Universal Robots PolyScope program: IAC002 PathMove.urp

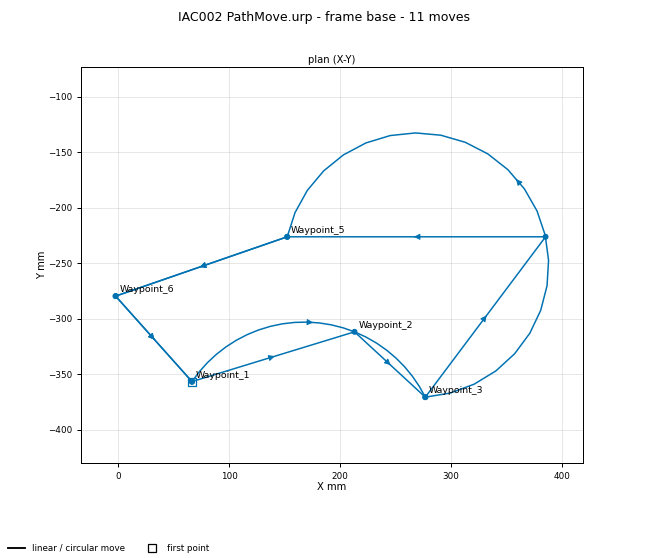
[picture p0: tool path of IAC002 PathMove.urp in frame base, 11 of 13 moves have a stored position in this frame; points joined in program order, loops and branches not executed]
Program IAC002 PathMove (installation=default directory=/programs createdIn=5.9.1.1031110 lastSavedIn=5.9.1.1031110 robotSerialNumber=20195501059)
Calibrated DH parameters: a=[0.000146, -0.418764, -0.053981, 0.000058, -0.000023, 0]; d=[0.162545, 37.319448, -206.067439, 168.881546, 0.09955, 0.099464]; alpha=[1.57004, -0.001979, 0.002304, 1.570607, -1.57066, 0]; deltaTheta=[0, -0.174616, -1.258233, 1.432844, -0.000001, 0]
Robot Program (runOnlyOnce=false)
  MoveP speed 100 mm/s, acceleration 1200 mm/s^2 (blendRadius=0.025 useActiveTCP=true) feature=Base
    Waypoint Waypoint_1: TCP in base x=66.517 y=-356.748 z=9.401 mm, rx=0.8699 ry=3.0055 rz=-0.0545 rad; joints [78.529, -92.143, 143.844, -143.739, 270.633, 20.88] deg; TCP offset x=0 y=0 z=174 mm, rx=0 ry=0 rz=0 rad
    Waypoint Waypoint_2: TCP in base x=212.953 y=-311.931 z=9.413 mm, rx=0.8699 ry=3.0054 rz=-0.0546 rad; joints [103.909, -89.736, 141.52, -143.858, 269.699, 46.246] deg
    Waypoint Waypoint_3: TCP in base x=276.697 y=-370.783 z=9.413 mm, rx=0.8699 ry=3.0055 rz=-0.0545 rad; joints [110.314, -78.862, 128.784, -141.938, 269.445, 52.645] deg
    Waypoint Waypoint_4: TCP in base x=385.033 y=-226.321 z=9.405 mm, rx=0.8698 ry=3.0055 rz=-0.0546 rad; joints [133, -80.507, 130.77, -141.882, 268.715, 75.321] deg
    Waypoint Waypoint_5: TCP in base x=152.305 y=-226.334 z=9.423 mm, rx=0.8699 ry=3.0055 rz=-0.0546 rad; joints [94.734, -109.57, 155.879, -138.422, 270.064, 37.053] deg
    Waypoint Waypoint_6: TCP in base x=-2.245 y=-279.765 z=9.416 mm, rx=0.8699 ry=3.0055 rz=-0.0546 rad; joints [59.76, -108.29, 155.126, -138.596, 271.286, 2.1] deg
    Waypoint Waypoint_1: TCP in base x=66.517 y=-356.748 z=9.401 mm, rx=0.8699 ry=3.0055 rz=-0.0545 rad; joints [78.529, -92.143, 143.844, -143.739, 270.633, 20.88] deg
  MoveP speed 150 mm/s, acceleration 1200 mm/s^2 (blendRadius=0.025 useActiveTCP=true) feature=Base
    CircleMove (OrientationMode=FIXED)
      Waypoint Waypoint_2: TCP in base x=212.953 y=-311.931 z=9.413 mm, rx=0.8699 ry=3.0054 rz=-0.0546 rad; joints [103.909, -89.736, 141.52, -143.858, 269.699, 46.246] deg
      Waypoint Waypoint_3: TCP in base x=276.697 y=-370.783 z=9.413 mm, rx=0.8699 ry=3.0055 rz=-0.0545 rad; joints [110.314, -78.862, 128.784, -141.938, 269.445, 52.645] deg
    CircleMove (OrientationMode=UNCONSTRAINED)
      Waypoint Waypoint_4: TCP in base x=385.033 y=-226.321 z=9.405 mm, rx=0.8698 ry=3.0055 rz=-0.0546 rad; joints [133, -80.507, 130.77, -141.882, 268.715, 75.321] deg
      Waypoint Waypoint_5: TCP in base x=152.305 y=-226.334 z=9.423 mm, rx=0.8699 ry=3.0055 rz=-0.0546 rad; joints [94.734, -109.57, 155.879, -138.422, 270.064, 37.053] deg
    Waypoint Waypoint_6: TCP in base x=-2.245 y=-279.765 z=9.416 mm, rx=0.8699 ry=3.0055 rz=-0.0546 rad; joints [59.76, -108.29, 155.126, -138.596, 271.286, 2.1] deg
  MoveL speed 250 mm/s, acceleration 1200 mm/s^2 (useActiveTCP=true) feature=Base
    Waypoint Waypoint_1: TCP in base x=66.517 y=-356.748 z=9.401 mm, rx=0.8699 ry=3.0055 rz=-0.0545 rad; joints [78.529, -92.143, 143.844, -143.739, 270.633, 20.88] deg
